TYPE ST_WorkTime :
STRUCT
	hours	: UDINT;
	minuts	: UINT;
	seconds	: UINT;
END_STRUCT
END_TYPE

(* stored: Version 1.1.0.1, ProductVersion 3.1.4024.12
   DUT ST_WorkTime: Id {a47abd02-c805-4524-8b6f-66147f9de5d3} *)
